(*
SerialCom_InfoSys_Sample1 (v2.0)
This sample sends and receives a string via serial communication.
Three hardware interfaces are used: Pc COM port, EL terminal, KL terminal
*)
PROGRAM SerialCommunicationHandler_1
VAR
	//fbEL6001	: FB_SerialCom;
	
	fbAsciiComm: FB_SerialCom;
	

	ReceiveStep: INT;
	ProcessVariableRead : BOOL;
	SetpointRead : BOOL;
	ProcessVariableReceived : BOOL;
	SetpointReceived : BOOL;
	SendStep: INT;
	pumpPressureStartSend: BOOL;
	start3: BOOL;
	received3: BOOL;
	start4: BOOL;
	received4: BOOL;
	Setpoint: STRING;
	
	fbUpdatePressureSetpoint: FB_UpdateSetpoint;
	pumpingPressureMeasurement: DINT;
	pumpingPressureSetpoint: DINT;
	pumpingPressureSetSetpoint: DINT;
	pumpingPressureSetSetpointPrev: DINT;
	tonMessageUpdate: TON;
	rTrigMessageNotUpdated: R_TRIG;
	OutputPowerRead: BOOL;
	OutputPowerReceived: BOOL;
	pumpingPressureOutputPower: DINT;
	testi: BOOL;
	flowMeasurement: DINT;
	preHeaterTemperatureMeasurement: DINT;
	preHeaterTemperatureSetpoint: DINT;
	preHeaterTemperatureOutputPower: DINT;
	fbUpdatePreHeaterTemperatureSetpoint: FB_UpdateSetpoint;
	preHeaterTemperatureSetSetpoint: DINT;
	preHeaterTemperatureSetSetpointPrev: DINT;
	preHeaterTemperatureStartSend: BOOL;
	separatorTemperatureMeasurement: DINT;
	separatorTemperatureSetpoint: DINT;
	separatorTemperatureOutputPower: DINT;
	fbUpdateSeparatorTemperatureSetpoint: FB_UpdateSetpoint;
	separatorTemperatureStartSend: BOOL;
	separatorTemperatureSetSetpoint: DINT;
	separatorTemperatureSetSetpointPrev: DINT;
	
	pumpingPressureSentSetpoint : DINT;
	ReactorPressureSetpoint: DINT;
END_VAR

// Receive data from controller
fbAsciiComm(TxBuffer:=TxBufferEL, RxBuffer:=RxBufferEL);
CASE ReceiveStep OF
	0: 
		// On startup: start data receiving
		//ProcessVariableRead := TRUE;
		ReceiveStep := 1;
	1:
		// Read pressure measurement from controller
		fbAsciiComm.StartSend(SendStringIn := 'L2M?*', start := TRUE);
		IF fbAsciiComm.Received THEN
			pumpingPressureMeasurement := F_AsciiNumberConvert(fbAsciiComm.sReceivedString);  
			fbAsciiComm.StopSend(stop := TRUE);
			ReceiveStep := 2;
		END_IF
	2:
		// Read pressure setpoint value
		fbAsciiComm.StartSend(SendStringIn := 'L2S?*', start := TRUE);
		IF fbAsciiComm.Received THEN
			pumpingPressureSetpoint := F_AsciiNumberConvert(fbAsciiComm.sReceivedString); 
			fbAsciiComm.StopSend(stop := TRUE);
			ReceiveStep := 3;
		END_IF		
	3:
		// Read pressure controller output power
		fbAsciiComm.StartSend(SendStringIn := 'L2W?*', start := TRUE);
		IF fbAsciiComm.Received THEN
			pumpingPressureOutputPower := F_AsciiNumberConvert(fbAsciiComm.sReceivedString); 
			fbAsciiComm.StopSend(stop := TRUE);
			ReceiveStep := 4;
		END_IF
	4:
		// Read flow measurement from controller
		fbAsciiComm.StartSend(SendStringIn := 'L3M?*', start := TRUE);
		IF fbAsciiComm.Received THEN
			flowMeasurement := F_AsciiNumberConvert(fbAsciiComm.sReceivedString);  
			fbAsciiComm.StopSend(stop := TRUE);
			ReceiveStep := 5;
		END_IF
	5:
		// Read preheater measurement from controller
		fbAsciiComm.StartSend(SendStringIn := 'L4M?*', start := TRUE);
		IF fbAsciiComm.Received THEN
			preHeaterTemperatureMeasurement := F_AsciiNumberConvert(fbAsciiComm.sReceivedString);  
			fbAsciiComm.StopSend(stop := TRUE);
			ReceiveStep := 6;
		END_IF
	6:
		// Read preheater setpoint value
		fbAsciiComm.StartSend(SendStringIn := 'L4S?*', start := TRUE);
		IF fbAsciiComm.Received THEN
			preHeaterTemperatureSetpoint := F_AsciiNumberConvert(fbAsciiComm.sReceivedString); 
			fbAsciiComm.StopSend(stop := TRUE);
			ReceiveStep := 7;
		END_IF		
	7:
		// Read preheater controller output power
		fbAsciiComm.StartSend(SendStringIn := 'L4W?*', start := TRUE);
		IF fbAsciiComm.Received THEN
			preHeaterTemperatureOutputPower := F_AsciiNumberConvert(fbAsciiComm.sReceivedString); 
			fbAsciiComm.StopSend(stop := TRUE);
			ReceiveStep := 8;
		END_IF	
	8:
		// Read separator measurement from controller
		fbAsciiComm.StartSend(SendStringIn := 'L5M?*', start := TRUE);
		IF fbAsciiComm.Received THEN
			separatorTemperatureMeasurement := F_AsciiNumberConvert(fbAsciiComm.sReceivedString);  
			fbAsciiComm.StopSend(stop := TRUE);
			ReceiveStep := 9;
		END_IF
	9:
		// Read separator setpoint value
		fbAsciiComm.StartSend(SendStringIn := 'L5S?*', start := TRUE);
		IF fbAsciiComm.Received THEN
			separatorTemperatureSetpoint := F_AsciiNumberConvert(fbAsciiComm.sReceivedString); 
			fbAsciiComm.StopSend(stop := TRUE);
			ReceiveStep := 10;
		END_IF		
	10:
		// Read separator controller output power
		fbAsciiComm.StartSend(SendStringIn := 'L5W?*', start := TRUE);
		IF fbAsciiComm.Received THEN
			separatorTemperatureOutputPower := F_AsciiNumberConvert(fbAsciiComm.sReceivedString); 
			fbAsciiComm.StopSend(stop := TRUE);
			ReceiveStep := 0;
		END_IF
			
END_CASE
tonMessageUpdate(IN:=NOT (fbAsciiComm.bStringReceived), PT := T#2S);
rTrigMessageNotUpdated(CLK := tonMessageUpdate.Q);
IF rTrigMessageNotUpdated.Q THEN
	fbAsciiComm.StopSend(stop := TRUE);
	ReceiveStep := 0;
END_IF

// Send data to controller

// Stop receiving data during send
IF pumpPressureStartSend OR preHeaterTemperatureStartSend OR separatorTemperatureStartSend THEN
	ReceiveStep := 0;
END_IF
// Update pressure setpoint
IF PressureControl.ReactorPressureAutoPID THEN
	pumpingPressureSentSetpoint := REAL_TO_DINT(PressureControl.ReactorPressurePIDcontrol.PIDy);
	PressureControl.ReactorPressurePIDcontrol.PIDy;
ELSE
	pumpingPressureSentSetpoint :=  pumpingPressureSetSetpoint;
END_IF
fbUpdatePressureSetpoint(fbAsciiComm := fbAsciiComm, bStartSend := pumpPressureStartSend, sParameterCharacter := 'S', iValue := pumpingPressureSentSetpoint, iSlaveNo := 2);
IF pumpingPressureSentSetpoint <> pumpingPressureSetSetpointPrev THEN
	pumpPressureStartSend := TRUE;
	fbAsciiComm.StopSend(stop := TRUE);
	pumpingPressureSetSetpointPrev := pumpingPressureSentSetpoint;
	//ReceiveStep := 2;
END_IF
// Update preheater temperature setpoint
fbUpdatePreHeaterTemperatureSetpoint(fbAsciiComm := fbAsciiComm, bStartSend := preHeaterTemperatureStartSend, sParameterCharacter := 'S', iValue := preHeaterTemperatureSetSetpoint, iSlaveNo := 4);
IF preHeaterTemperatureSetSetpoint <> preHeaterTemperatureSetSetpointPrev THEN
	preHeaterTemperatureStartSend := TRUE;
	fbAsciiComm.StopSend(stop := TRUE);
	preHeaterTemperatureSetSetpointPrev := preHeaterTemperatureSetSetpoint;
	//ReceiveStep := 6;
END_IF
// Update preheater temperature setpoint
fbUpdateSeparatorTemperatureSetpoint(fbAsciiComm := fbAsciiComm, bStartSend := separatorTemperatureStartSend, sParameterCharacter := 'S', iValue := separatorTemperatureSetSetpoint, iSlaveNo := 5);
IF separatorTemperatureSetSetpoint <> separatorTemperatureSetSetpointPrev THEN
	separatorTemperatureStartSend := TRUE;
	fbAsciiComm.StopSend(stop := TRUE);
	separatorTemperatureSetSetpointPrev := separatorTemperatureSetSetpoint;
	//ReceiveStep := 10;
END_IF

END_PROGRAM

(* stored: Version 1.1.0.1, ProductVersion 3.1.4024.9
   POU SerialCommunicationHandler_1: Id {e27a22ad-5f01-4f89-9a8a-8e29e3fb8faf}, SpecialFunc None *)
